// TIA Portal V17 export
// export: Created 2023-04-11T09:33:30.9672072Z, ExportSetting WithDefaults, DisplayName Totally Integrated Automation Portal, DisplayVersion V17 Update 3, DisplayName TIA Portal Openness, DisplayVersion V17 Update 3, DisplayName TIA Portal Version Control Interface, DisplayVersion V17, DisplayName SINAMICS Startdrive Advanced, DisplayVersion V17 Update2, DisplayName SINAMICS Startdrive G130, G150, S120, S150, SINAMICS MV, S210, DisplayVersion V17 Update2, DisplayName SINAMICS Startdrive G110M, G120, G120C, G120D, G120P, G115D, DisplayVersion V17 Update2, DisplayName STEP 7 Professional, DisplayVersion V17 Update 3, DisplayName STEP 7 Safety, DisplayVersion V17, DisplayName WinCC UA Professional, DisplayVersion V17 Update 3
FUNCTION_BLOCK "FB_faultModule"   // FB21001, LAD
{ S7_Optimized_Access := 'TRUE' }
VERSION : 0.1
// stored: AutoNumber false, IsIECCheckEnabled false, IsRetainMemResEnabled false, MemoryReserve 100, SetENOAutomatically false, UDAEnableTagReadback false
   VAR_INPUT
      Double_Coil : Bool;
      Coil_A : Bool;
      Coil_B : Bool;
      Sensor_A : Bool;
      With_A : Bool;
      Sensor_B : Bool;
      With_B : Bool;
      Monitoring_On : Bool;
      TimeForMovement_A : Time;
      TimeForMovement_B : Time;
   END_VAR
   VAR_OUTPUT
      Error_WP : Bool;
      Error_HP : Bool;
   END_VAR
   VAR
      FaultHM_WP : Bool;
      FaultHM_HP : Bool;
      P_Flank : Bool;
      WPTime { S7_SetPoint := 'True'} : TON_TIME;
      HPTime { S7_SetPoint := 'True'} : TON_TIME;
   END_VAR
BEGIN

REGION Network 1
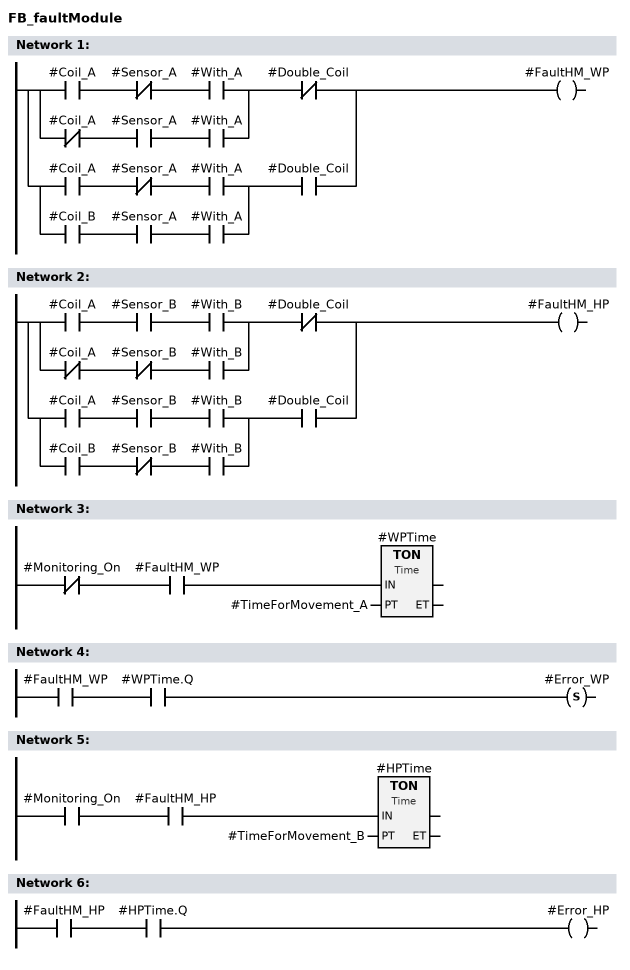
   RUNG wire#powerrail
      Contact( #Coil_A )
      I_Contact( #Sensor_A )
      Contact( #With_A )
      wire#w1
      I_Contact( #Double_Coil )
      wire#w2
      Coil( #FaultHM_WP )
   END_RUNG
   RUNG wire#powerrail
      I_Contact( #Coil_A )
      Contact( #Sensor_A )
      Contact( #With_A )
   END_RUNG wire#w1
   RUNG wire#powerrail
      Contact( #Coil_A )
      I_Contact( #Sensor_A )
      Contact( #With_A )
      wire#w3
      Contact( #Double_Coil )
   END_RUNG wire#w2
   RUNG wire#powerrail
      Contact( #Coil_B )
      Contact( #Sensor_A )
      Contact( #With_A )
   END_RUNG wire#w3
   // the same network as SCL:
   #FaultHM_WP := (((#Coil_A AND NOT #Sensor_A AND #With_A) OR (NOT #Coil_A AND #Sensor_A AND #With_A)) AND NOT #Double_Coil) OR (((#Coil_A AND NOT #Sensor_A AND #With_A) OR (#Coil_B AND #Sensor_A AND #With_A)) AND #Double_Coil);
END_REGION

REGION Network 2
   RUNG wire#powerrail
      Contact( #Coil_A )
      Contact( #Sensor_B )
      Contact( #With_B )
      wire#w1
      I_Contact( #Double_Coil )
      wire#w2
      Coil( #FaultHM_HP )
   END_RUNG
   RUNG wire#powerrail
      I_Contact( #Coil_A )
      I_Contact( #Sensor_B )
      Contact( #With_B )
   END_RUNG wire#w1
   RUNG wire#powerrail
      Contact( #Coil_A )
      Contact( #Sensor_B )
      Contact( #With_B )
      wire#w3
      Contact( #Double_Coil )
   END_RUNG wire#w2
   RUNG wire#powerrail
      Contact( #Coil_B )
      I_Contact( #Sensor_B )
      Contact( #With_B )
   END_RUNG wire#w3
   // the same network as SCL:
   #FaultHM_HP := (((#Coil_A AND #Sensor_B AND #With_B) OR (NOT #Coil_A AND NOT #Sensor_B AND #With_B)) AND NOT #Double_Coil) OR (((#Coil_A AND #Sensor_B AND #With_B) OR (#Coil_B AND NOT #Sensor_B AND #With_B)) AND #Double_Coil);
END_REGION

REGION Network 3
   RUNG wire#powerrail
      I_Contact( #Monitoring_On )
      Contact( #FaultHM_WP )
      { S7_Templates := "time_type := Time" } #WPTime.TON(pt := #TimeForMovement_A, et =>)
   END_RUNG
   // the same network as SCL:
   #WPTime(IN := NOT #Monitoring_On AND #FaultHM_WP, PT := #TimeForMovement_A);   // TON
END_REGION

REGION Network 4
   RUNG wire#powerrail
      Contact( #FaultHM_WP )
      Contact( #WPTime.Q )
      S_Coil( #Error_WP )
   END_RUNG
   // the same network as SCL:
   IF #FaultHM_WP AND #WPTime.Q THEN #Error_WP := TRUE; END_IF;
END_REGION

REGION Network 5
   RUNG wire#powerrail
      Contact( #Monitoring_On )
      Contact( #FaultHM_HP )
      { S7_Templates := "time_type := Time" } #HPTime.TON(pt := #TimeForMovement_B, et =>)
   END_RUNG
   // the same network as SCL:
   #HPTime(IN := #Monitoring_On AND #FaultHM_HP, PT := #TimeForMovement_B);   // TON
END_REGION

REGION Network 6
   RUNG wire#powerrail
      Contact( #FaultHM_HP )
      Contact( #HPTime.Q )
      Coil( #Error_HP )
   END_RUNG
   // the same network as SCL:
   #Error_HP := #FaultHM_HP AND #HPTime.Q;
END_REGION
END_FUNCTION_BLOCK
